{attribute 'linkalways'} 
{attribute 'no_explicit_call' := 'This FB is a CLASS and must be accessed using methods or properties'}
{attribute 'enable_dynamic_creation'}
FUNCTION_BLOCK FINAL SEL_SINT EXTENDS Node
VAR
	g : _BOOL(FALSE);
	in1 : _SINT(0);
	in2 : _SINT(0);
	out : _SINT(0);
END_VAR

METHOD PUBLIC Clone : I_Node
VAR
	pNode : POINTER TO SEL_SINT;
END_VAR
pNode := __NEW(SEL_SINT);
Clone := pNode^;
END_METHOD

METHOD FB_init : BOOL
VAR_INPUT
	bInitRetains : BOOL; // if TRUE, the retain variables are initialized (warm start / cold start)
	bInCopyCode : BOOL;  // if TRUE, the instance afterwards gets moved into the copy code (online change)
END_VAR
AddInput('g',THIS^.g);
AddInput('in1',THIS^.in1);
AddInput('in2',THIS^.in2);
AddOutput('out', THIS^.out);
END_METHOD

METHOD PROTECTED OnExecute
VAR
END_VAR
IF g.value THEN
	out.value := in2.value;
ELSE
	out.value := in1.value;
END_IF
END_METHOD

END_FUNCTION_BLOCK

(* stored: Version 1.1.0.1, ProductVersion 3.1.4024.15
   POU SEL_SINT: Id {b70fab52-257c-4b67-bba0-4d28ceff1d7f}, SpecialFunc None
   Folder Constructor: Id {95b88e4d-563b-4819-8414-9d7393807870}
   Method Clone: Id {492b56e3-e739-4a43-aa72-537b1ebcbadb}
   Method FB_init: Id {c7a54d94-6029-4186-85f3-8d9fb987e1a2}
   Method OnExecute: Id {2b862612-8cfe-42e2-a8ec-dbf94dc9ad84} *)
